Fanuc KAREL source: FRAME__3.kl

PROGRAM T
%NOLOCKGROUP
VAR
 v0 : POSITION
 v1 : POSITION
 v2 : POSITION
 res : POSITION
BEGIN
 res = FRAME(v0, v1, v2)
END T
